# EPICS autosave request: iocBoot/obsolete/ioc13bmd/auto_positions.req
file "CARS_88_motor_positions.req", P=$(P)
file "CARS_motor_positions.req",         P=$(P), M=m105
file "CARS_motor_positions.req",         P=$(P), M=m106
file "CARS_motor_positions.req",         P=$(P), M=m107
file "CARS_motor_positions.req",         P=$(P), M=m108
file "CARS_motor_positions.req",         P=$(P), M=m109
file "CARS_motor_positions.req",         P=$(P), M=m110
file "CARS_motor_positions.req",         P=$(P), M=m111
file "CARS_motor_positions.req",         P=$(P), M=m112
